TYPE ST_AnalogInputData :
STRUCT
	Value			: INT;
	Status			: ST_AnalogInputDiag;
END_STRUCT
END_TYPE

(* stored: Version 1.1.0.1, ProductVersion 3.1.4026.18
   DUT ST_AnalogInputData: Id {b966fc4e-5f05-491f-9b79-9af3a9645c60} *)
